{attribute 'qualified_only'}
{attribute 'strict'}
TYPE E_TimeSource :
(
	FileTime := 0,
	DcTaskInfo := 1,
	fbLocalSystemTime := 2
);
END_TYPE

(* stored: Version 1.1.0.1, ProductVersion 3.1.4024.12
   DUT E_TimeSource: Id {e5429833-6cda-4ee6-a471-89d230ee4341} *)
